(* IEC 61131-3 sources: CodesysTest/alpha/export/FBs/Components/Motors/Applied Motion/FB_AppliedMotionStepServoEIPPassthrough.pou, 2 files *)

(* ---- DoneClamping.m.st ---- *)
(*#-#-#-#-#-#-#-#-#-#---Declaration---#-#-#-#-#-#-#-#-#-#-#-#-#*)

METHOD DoneClamping
VAR_INPUT
END_VAR
(*#-#-#-#-#-#-#-#-#-#---Implementation---#-#-#-#-#-#-#-#-#-#-#-#-#*)

sclCommand := 16#434D; // CM Control Mode
parameter1 := 21;

commandSuccessful := FALSE;
commands.SendHostCommand := TRUE;

(* ---- SetPositionFaultLimit.m.st ---- *)
(*#-#-#-#-#-#-#-#-#-#---Declaration---#-#-#-#-#-#-#-#-#-#-#-#-#*)

METHOD SetPositionFaultLimit
VAR_INPUT
	positionLimit : DINT;
END_VAR
(*#-#-#-#-#-#-#-#-#-#---Implementation---#-#-#-#-#-#-#-#-#-#-#-#-#*)

sclCommand := 16#5046; // PF (Position Fault)
parameter1 := positionLimit;

commandSuccessful := FALSE;
commands.SendHostCommand := TRUE;
